FUNCTION_BLOCK DualHysteresis (* 2-way conversion of Analog to Digital with Hysteresis *)
  (* Standard: 61499-2; Description: Copyright (c) 2023 HR Agrartechnik GmbH This program and the accompanying materials are made available under the terms of the Eclipse Public License 2.0 which is available at https://www.eclipse.org/legal/epl-2.0/ SPDX-License-Identifier: EPL-2.0 *)
  (* Version 3.0, 2025-04-14, Patrick Aigner, changed package *)
  (* Version 1.0, 2023-06-06, Franz Höpfinger, HR Agrartechnik GmbH *)
  PACKAGE eclipse4diac::signalprocessing;
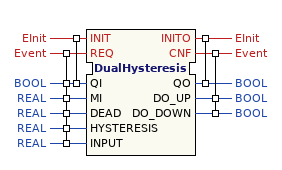
  EVENT_INPUT
    INIT : EInit WITH QI; (* Initialization Request *)
    REQ WITH QI, MI, DEAD, INPUT, HYSTERESIS; (* Normal Execution Request *)
  END_EVENT
  EVENT_OUTPUT
    INITO : EInit WITH QO; (* Initialization Confirm *)
    CNF WITH DO_UP, DO_DOWN; (* Execution Confirmation *)
  END_EVENT
  VAR_INPUT
    QI : BOOL; (* Input event qualifier *)
    MI : REAL := 0.5; (* MID Setting can e.g. be 0.5 meaning 50% *)
    DEAD : REAL := 0.1; (* Deadband around MID can be e.g. 0.1 meaning 10% *)
    HYSTERESIS : REAL := 0.1; (* Hysteresis can be 0.1 meaning 10% *)
    INPUT : REAL; (* Value *)
  END_VAR
  VAR_OUTPUT
    QO : BOOL;
    DO_UP : BOOL; (* UP *)
    DO_DOWN : BOOL; (* DOWN *)
  END_VAR
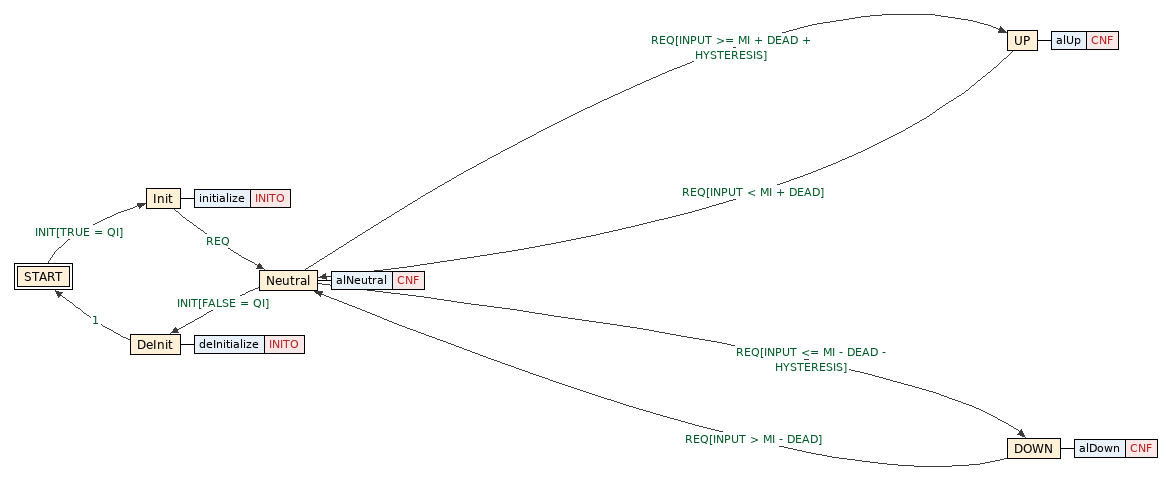
  EC_STATES
    START; (* Initial State *)
    Init : initialize -> INITO; (* Initialization *)
    UP : alUp -> CNF; (* Normal execution *)
    Neutral : alNeutral -> CNF;
    DeInit : deInitialize -> INITO;
    DOWN : alDown -> CNF;
  END_STATES
  EC_TRANSITIONS
    START TO Init := INIT[TRUE = QI];
    Init TO Neutral := REQ;
    Neutral TO DeInit := INIT[FALSE = QI];
    Neutral TO UP := REQ[INPUT >= MI + DEAD + HYSTERESIS];
    DeInit TO START := 1;
    Neutral TO DOWN := REQ[INPUT <= MI - DEAD - HYSTERESIS];
    DOWN TO Neutral := REQ[INPUT > MI - DEAD];
    UP TO Neutral := REQ[INPUT < MI + DEAD];
  END_TRANSITIONS
  ALGORITHM initialize IN ST:
QO := QI;
(* in any case go safe State *)
DO_UP := BOOL#FALSE;
DO_DOWN := BOOL#FALSE;
  END_ALGORITHM
  ALGORITHM deInitialize IN ST:
QO := BOOL#FALSE;
(* in any case go safe State *)
DO_UP := BOOL#FALSE;
DO_DOWN := BOOL#FALSE;
  END_ALGORITHM
  ALGORITHM alNeutral IN ST:
QO := QI;
(* in any case go safe State *)
DO_UP := BOOL#FALSE;
DO_DOWN := BOOL#FALSE;
  END_ALGORITHM
  ALGORITHM alUp IN ST:
QO := QI;
IF TRUE = QI THEN
	(* only perform normal operation of QI is true *)
	DO_UP := BOOL#TRUE;
	DO_DOWN := BOOL#FALSE;
END_IF;
  END_ALGORITHM
  ALGORITHM alDown IN ST:
QO := QI;
IF TRUE = QI THEN
	(* only perform normal operation of QI is true *)
	DO_UP := BOOL#FALSE;
	DO_DOWN := BOOL#TRUE;
END_IF;
  END_ALGORITHM
END_FUNCTION_BLOCK
